// TIA Portal V19 export
TYPE "lexchangetray_typeUnEmnTranserfCondition"
// Type: Bool
// stored: Access Published
   STRUCT
      axisPosMoveCondition : Bool;   // Manual mode parameters for axis control interface
   END_STRUCT;
END_TYPE
